FUNCTION_BLOCK FB_LoadingSequence
VAR_INPUT
END_VAR
VAR_OUTPUT
END_VAR
VAR
END_VAR

END_FUNCTION_BLOCK

(* stored: Version 1.1.0.1, ProductVersion 3.1.4026.18
   POU FB_LoadingSequence: Id {1353c084-c4cd-44a2-a00e-480bb357bf7f}, SpecialFunc None *)
